(*
Nazwa:			S_RFIDCheck
Opis:			sprawdzanie RFID
Wersja:			v0.1
Data:			2024-12-03
Autor:			
Urzadzenia:		
Konfiguracja:	
Info:

*)
TYPE S_RFIDCheck :
STRUCT 
	iNumber				: INT;		//Numer RFID	
	iReaded1			: INT;		//Odczytano z czytnika nr 1
	iReaded2			: INT;		//Odczytano z czytnika nr 2
	iReaded3			: INT;		//Odczytano z czytnika nr 3
	iReaded4			: INT;		//Odczytano z czytnika nr 4
	iReaded5			: INT;		//Odczytano z czytnika nr 5
END_STRUCT
END_TYPE

(* stored: Version 1.1.0.1, ProductVersion 3.1.4026.13, FileIdentifier 498a9133668e89558660b46add8f2698febef673, FileSignature 01739d768da4b355edec8de5481e744a62f053d9b17950e75549691048896f267c54dda5451aca0122c293a0d3d5f949fb8a0632d9cd774e4ec7c286454af0e1fd14931568e8f3742fe384d75f614ef87596847dbe18cd84e088f2492f9c708aa70d852cfa60e42199235b9d57e231a25852886e0b4980cca825862ae6f52157cb89aa31d09aa8cc22dffdeb635ac973a9b2b5e48fc47836e34ad86e56e5dd4974388694975929aa07c120c99c22337ef8ca3b27a530d309da879b2a9f963ca773efd3339d2ea316e1c9cf09c8f831c7c74c6ad9eac69bce69362cf3a597e3802108b07edf5c8ce1a0486237c07c81f683e3bb5b0c9c52c294c25d3c96680c09
   DUT S_RFIDCheck: Id {ddeb7dbc-54e0-45d1-9873-65e3bafa87ee} *)
